FUNCTION_BLOCK ElapsedTimeBasic (* Basic Function Block Type *)
  (* Standard: 61499-2 *)
  (* Version 0.0, 7/7/2026, Schneider Electric, Template *)
  PACKAGE SE.Nereda;
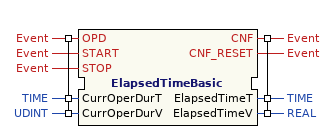
  EVENT_INPUT
    OPD WITH CurrOperDurT, CurrOperDurV; (* Normal Execution Request *)
    START;
    STOP;
  END_EVENT
  EVENT_OUTPUT
    CNF WITH ElapsedTimeT, ElapsedTimeV; (* Execution Confirmation *)
    CNF_RESET;
  END_EVENT
  VAR_INPUT
    CurrOperDurT : TIME; (* Input event qualifier *)
    CurrOperDurV : UDINT;
  END_VAR
  VAR_OUTPUT
    ElapsedTimeT : TIME; (* Output event qualifier *)
    ElapsedTimeV : REAL;
  END_VAR
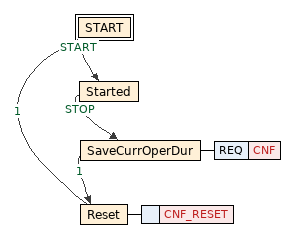
  EC_STATES
    START; (* Initial State *)
    Started;
    SaveCurrOperDur : REQ -> CNF;
    Reset : -> CNF_RESET;
  END_STATES
  EC_TRANSITIONS
    START TO Started := START;
    Started TO SaveCurrOperDur := STOP;
    SaveCurrOperDur TO Reset := 1;
    Reset TO START := 1;
  END_TRANSITIONS
  ALGORITHM REQ IN ST: (* Normally executed algorithm *)
;
ElapsedTimeT := CurrOperDurT;
ElapsedTimeV := UDINT_TO_REAL(CurrOperDurV) * 1000;
  END_ALGORITHM
END_FUNCTION_BLOCK
